// TIA Portal V19 export
TYPE "PPrf_SetUp_Aut"
// stored: Access Published
   STRUCT
      Rollformer : Struct   // Profilatrice - Posizione assi di regolazione formato
         Passaggio02_OP : Real;   // Roll Stand 02 OP. Side / Passaggio 02 Lato OP - Posizione (mm) per lavoro NERVATURA
         Passaggio02_MOT : Real;   // Roll Stand 02 MOT. Side / Passaggio 02 Lato MOT - Posizione (mm) per lavoro NERVATURA
         Passaggio14_OP : Real;
         Passaggio14_MOT : Real;
         Passaggio17_OP : Real;
         Passaggio17_MOT : Real;
         Passaggio18_OP : Real;
         Passaggio18_MOT : Real;
         Cassetta_1_OP : Real;   // Roll Stand Frame / Spalla OP - Posizione (mm)
         Cassetta_1_MOT : Real;   // Roll Stand Frame / Spalla MOT - Posizione (mm)
         Cassetta_2_OP : Real;   // Roll Stand Frame / Spalla OP - Posizione (mm)
         Cassetta_2_MOT : Real;   // Roll Stand Frame / Spalla MOT - Posizione (mm)
         Cassetta_3_OP : Real;   // Roll Stand Frame / Spalla OP - Posizione (mm)
         Cassetta_3_MOT : Real;   // Roll Stand Frame / Spalla MOT - Posizione (mm)
      END_STRUCT;
      Bordatrice : Struct   // Macchina chiusra bordi
         Passaggio01_L : Real;   // Roll Stand / Passaggio 01 SINISTRA - Posizione (mm)
         Passaggio01_R : Real;   // Roll Stand / Passaggio 01 DESTRA - Posizione (mm)
         Passaggio02_L : Real;   // Roll Stand / Passaggio 02 SINISTRA - Posizione (mm)
         Passaggio02_R : Real;   // Roll Stand / Passaggio 02 DESTRA - Posizione (mm)
         Passaggio03_L : Real;   // Roll Stand / Passaggio 03 SINISTRA - Posizione (mm)
         Passaggio03_R : Real;   // Roll Stand / Passaggio 03 DESTRA - Posizione (mm)
         Passaggio04_L : Real;   // Roll Stand / Passaggio 04 SINISTRA - Posizione (mm)
         Passaggio04_R : Real;   // Roll Stand / Passaggio 04 DESTRA - Posizione (mm)
         Cassetta_1_OP : Real;   // Cassetta 1 Operatore - Posizione (mm)
      END_STRUCT;
   END_STRUCT;
END_TYPE
